(* PLC project Unnamed, Unknown Unnamed 1 *)
(* stored: creationDateTime 2024-01-27T21:00:33, modificationDateTime 2024-01-29T10:59:28 *)

PROGRAM PreTreatment
  VAR
    P201 AT %QX0.0 : BOOL;
    P202 AT %QX0.1 : BOOL;
    P203 AT %QX0.2 : BOOL;
    P204 AT %QX0.3 : BOOL;
    P205 AT %QX0.4 : BOOL;
    P206 AT %QX0.5 : BOOL;
    MV201 AT %QX0.6 : BOOL;
    LS201 AT %QW0 : INT;
    LS202 AT %QW1 : INT;
  END_VAR

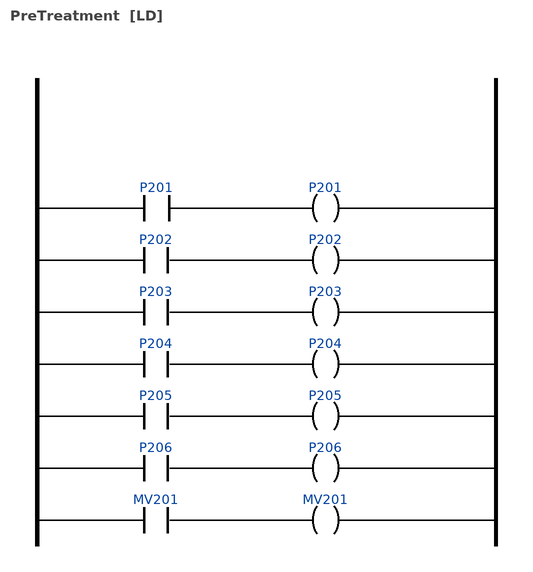
(* LD diagram, written out as Structured Text *)
P201 := P201;
P202 := P202;
P203 := P203;
P204 := P204;
P205 := P205;
P206 := P206;
MV201 := MV201;
END_PROGRAM

CONFIGURATION Config0
  RESOURCE Res0 ON PLC
    TASK task0(INTERVAL := T#20ms, PRIORITY := 0);
    PROGRAM instance0 WITH task0 : PreTreatment;
  END_RESOURCE
END_CONFIGURATION
